FUNCTION_BLOCK AR_CALIBRATE_SQ_REF (* Adapter-based sequential two-point calibration (offset then scale) with ECC-enforced order - reference targets (Y_Offset/Y_Scale) are live AR sockets, persisted via 2 additional AR2 plugs (ZERO/SPAN) *)
  (* Standard: 61499-1 *)
  (* Version 1.0, 2026-08-31, Meisterschulen am Ostbahnhof *)
  PACKAGE adapter::Engineering::measurements;
  (* Documentation:
  Formula
    Y = (X + OFFSET) * SCALE Reference Targets (Y_Offset / Y_Scale) are live AR Sockets
   Unlike AR_CALIBRATE_SQ, the two target values are not plain InputVars set via a SET event - they are live AR Sockets (Y_Offset, Y_Scale), fed the same way as X (e.g. from an editable VT input field). Every time a new value arrives, it is immediately mirrored out through the new AR2 Plugs ZERO/SPAN so it can be persisted (INI_AR2 or NVS_AR2) exactly like OFFSET/SCALE already are.
   Important: exactly like OFFSET/SCALE, the CO/CS algorithms never read the raw incoming Y_Offset.D1/Y_Scale.D1 directly for their math - they read the round-tripped ZERO.DI1/SPAN.DI1 instead (the value echoed back by the external INI_AR2, which requires SETM=TRUE on that instance to actually echo). This keeps both reference values consistent with what's really persisted, and is what makes a boot-restored default usable without the operator having to re-enter it first.
   Calibration (Two-Point, ECC-Enforced)
    - Offset (CO): Apply low reference, set Y_Offset (ZERO) to desired output, trigger CO
   OFFSET := ZERO.DI1 / SCALE - X → after CO, Y always equals ZERO.DI1 (independent of SCALE)
   - Scale (CS): Apply high reference, set Y_Scale (SPAN) to desired output, trigger CS
   Calculates SCALE and OFFSET decoupled using both reference points (SPAN.DI1 and the CO-time ZERO.DI1) → after CS, the line passes exactly through both points
    Note: Both Y_Offset and Y_Scale are target values on the output side.
    - CS is only reachable after offset calibration (state WAIT_CS) – enforced by ECC
   - CO can be repeated at any time to re-calibrate offset
   - Normal calculation via X.E1 works in all states
  *)
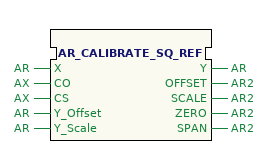
  SOCKETS
    X : adapter::types::unidirectional::AR; (* Raw Input *)
    CO : adapter::types::unidirectional::AX; (* Calibrate Offset *)
    CS : adapter::types::unidirectional::AX; (* Calibrate Scale *)
    Y_Offset : adapter::types::unidirectional::AR; (* Target output Y at low calibration point (ZERO), live input *)
    Y_Scale : adapter::types::unidirectional::AR; (* Target output Y at high calibration point (SPAN), live input *)
  END_SOCKETS
  PLUGS
    Y : adapter::types::unidirectional::AR; (* Calibrated Output *)
    OFFSET : adapter::types::bidirectional::AR2; (* Stored offset value (initial 0.0) *)
    SCALE : adapter::types::bidirectional::AR2; (* Stored scale value (initial 1.0) *)
    ZERO : adapter::types::bidirectional::AR2; (* Persisted low-point target reference (Y_Offset / Nullpunkt) *)
    SPAN : adapter::types::bidirectional::AR2; (* Persisted high-point target reference (Y_Scale / Spanne) *)
  END_PLUGS
  VAR
    X_LOW_INT : REAL; (* Stored raw value at CO *)
    Y_LOW_INT : REAL; (* Stored target value at CO *)
  END_VAR
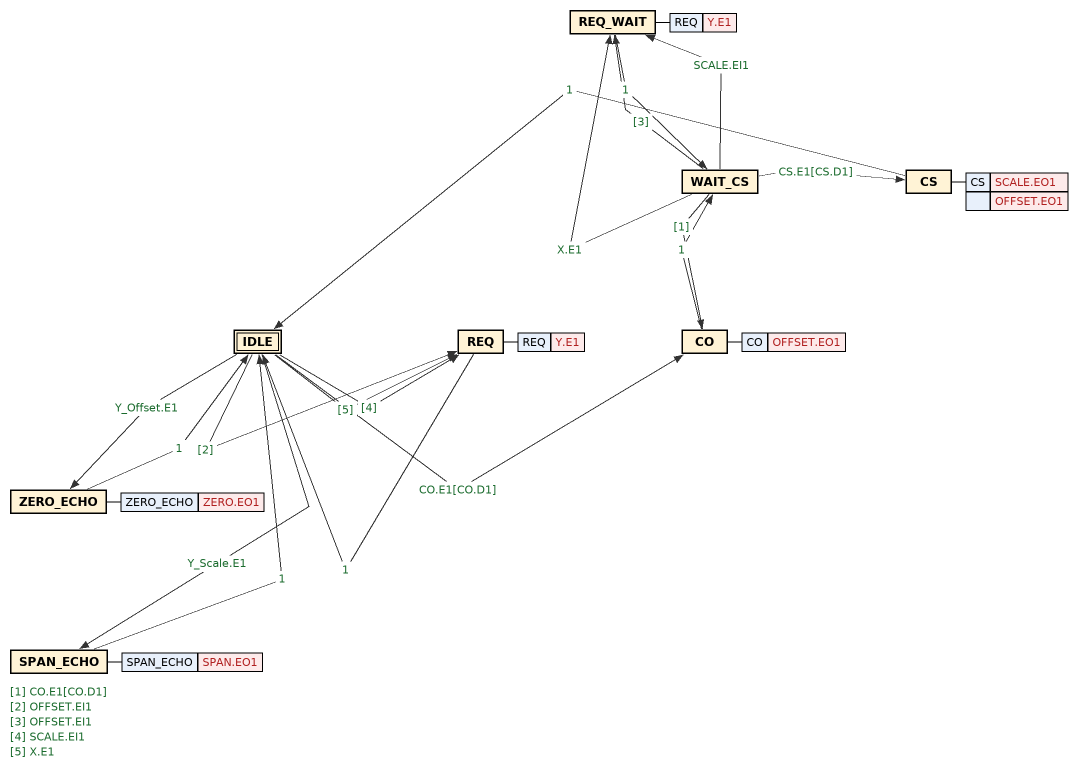
  EC_STATES
    IDLE;
    REQ : REQ -> Y.E1;
    CO : CO -> OFFSET.EO1;
    WAIT_CS;
    REQ_WAIT : REQ -> Y.E1;
    CS : CS -> SCALE.EO1, -> OFFSET.EO1;
    ZERO_ECHO : ZERO_ECHO -> ZERO.EO1;
    SPAN_ECHO : SPAN_ECHO -> SPAN.EO1;
  END_STATES
  EC_TRANSITIONS
    IDLE TO REQ := X.E1;
    REQ TO IDLE := 1;
    IDLE TO CO := CO.E1[CO.D1];
    CO TO WAIT_CS := 1;
    WAIT_CS TO REQ_WAIT := X.E1;
    REQ_WAIT TO WAIT_CS := 1;
    WAIT_CS TO CS := CS.E1[CS.D1];
    CS TO IDLE := 1;
    WAIT_CS TO CO := CO.E1[CO.D1];
    IDLE TO REQ := OFFSET.EI1;
    IDLE TO REQ := SCALE.EI1;
    WAIT_CS TO REQ_WAIT := OFFSET.EI1;
    WAIT_CS TO REQ_WAIT := SCALE.EI1;
    IDLE TO ZERO_ECHO := Y_Offset.E1;
    ZERO_ECHO TO IDLE := 1;
    IDLE TO SPAN_ECHO := Y_Scale.E1;
    SPAN_ECHO TO IDLE := 1;
  END_TRANSITIONS
  ALGORITHM REQ IN ST: (* REQ *)
(* calculate calibrated output *)
Y.D1 := (X.D1 + OFFSET.DI1) * SCALE.DI1;
  END_ALGORITHM
  ALGORITHM CO IN ST: (* CO *)
X_LOW_INT := X.D1;
Y_LOW_INT := ZERO.DI1;
IF SCALE.DI1 <> 0.0 THEN
	OFFSET.DO1 := ZERO.DI1 / SCALE.DI1 - X.D1;
ELSE
	OFFSET.DO1 := ZERO.DI1 - X.D1;
END_IF;
  END_ALGORITHM
  ALGORITHM CS IN ST: (* CS *)
IF (X.D1 - X_LOW_INT) <> 0.0 THEN
	SCALE.DO1 := (SPAN.DI1 - Y_LOW_INT) / (X.D1 - X_LOW_INT);
	IF SCALE.DO1 <> 0.0 THEN
		OFFSET.DO1 := Y_LOW_INT / SCALE.DO1 - X_LOW_INT;
	END_IF;
END_IF;
  END_ALGORITHM
  ALGORITHM ZERO_ECHO IN ST: (* Persist live Y_Offset reference (ZERO) to INI *)
ZERO.DO1 := Y_Offset.D1;
  END_ALGORITHM
  ALGORITHM SPAN_ECHO IN ST: (* Persist live Y_Scale reference (SPAN) to INI *)
SPAN.DO1 := Y_Scale.D1;
  END_ALGORITHM
END_FUNCTION_BLOCK
